PROGRAM YaxisBar
VAR
	Zero: MC_SetPosition;
	power: MC_Power;
	MC_MoveAbsolute: MC_MoveAbsolute;
	MC_Jog_0: MC_Jog;
	FB_CoEAX8000BrakeControl_0: FB_CoEAX8000BrakeControl;
	Release: BOOL;
	Brake: E_BrakeMode := eBrakeMode_Unlock;
	VeloLeading: MC_MoveAbsolute;
	bVeloStart: BOOL;
	R_TRIG_0: R_TRIG;
	
	Cutout			:bool;
	
	velolatch		at %I* : BOOL;
	F_trig_0: f_TRIG;
	
		VeloLOWCUT: UDINT;
	R_TRIG_1: R_TRIG;
	F_TRIG_1: F_TRIG;
	VeloHIGHCUT: UDINT;
	VeloMIDCUT: UDINT;
	SR1: SR;
	
	VeloStartPoint			:LREAL;
	VeloEndPoint			:LREAL;
	
END_VAR

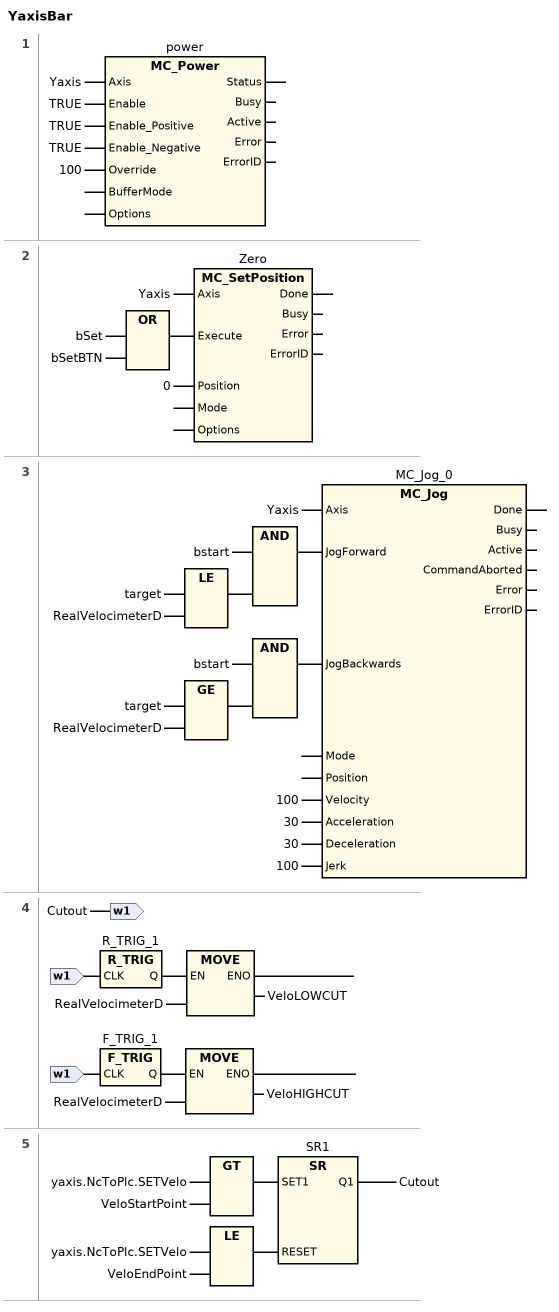
// NETWORK 1
power(Axis := Yaxis, Enable := TRUE, Enable_Positive := TRUE, Enable_Negative := TRUE, Override := 100); // MC_Power

// NETWORK 2
Zero(Axis := Yaxis, Execute := bSet OR bSetBTN, Position := 0); // MC_SetPosition

// NETWORK 3
MC_Jog_0(
    Axis := Yaxis,
    JogForward := bstart AND target <= RealVelocimeterD,
    JogBackwards := bstart AND target >= RealVelocimeterD,
    Velocity := 100,
    Acceleration := 30,
    Deceleration := 30,
    Jerk := 100); // MC_Jog

// NETWORK 4
R_TRIG_1(CLK := Cutout); // R_TRIG
IF R_TRIG_1.Q THEN VeloLOWCUT := RealVelocimeterD; END_IF
F_TRIG_1(CLK := Cutout); // F_TRIG
IF F_TRIG_1.Q THEN VeloHIGHCUT := RealVelocimeterD; END_IF

// NETWORK 5
SR1(SET1 := yaxis.NcToPlc.SETVelo > VeloStartPoint, RESET := yaxis.NcToPlc.SETVelo <= VeloEndPoint); // SR
Cutout := SR1.Q1;

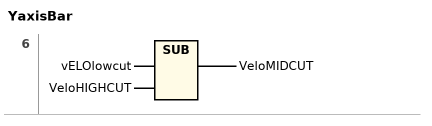
// NETWORK 6
VeloMIDCUT := vELOlowcut - VeloHIGHCUT;

END_PROGRAM

(* stored: Version 1.1.0.1, ProductVersion 3.1.4024.12
   POU YaxisBar: Id {5f9b8433-6e36-469a-a40a-3ad99166923e}, SpecialFunc None *)
